FUNCTION_BLOCK FB_ConveyerTimer
VAR_INPUT
END_VAR
VAR_OUTPUT
	bReadyToPlace : BOOL;
END_VAR
VAR
	velocityTime	: TON;
	bConveyerMovement: BOOL;
END_VAR

velocityTime(
	IN := bConveyerMovement,
	PT := T#0.2S
	);

IF GVL_Conveyer.ConveyerAxis.NcToPlc.SetVelo = 0 THEN
		bConveyerMovement := FALSE;
	ELSE
		bConveyerMovement := TRUE;
	END_IF

IF velocityTime.Q THEN
	bReadyToPlace := TRUE;
ELSE
	bReadyToPlace := FALSE;
END_IF

END_FUNCTION_BLOCK

(* stored: Version 1.1.0.1, ProductVersion 3.1.4024.11
   POU FB_ConveyerTimer: Id {93d6b353-6e10-4ea1-b929-36aa8af36d9d}, SpecialFunc None *)
